Fanuc KAREL source: kb00125.KL

PROGRAM KB00125
%STACKSIZE=65535
%PRIORITY=65535
%NOLOCKGROUP
VAR
P1 : STRING[80]
P2 : INTEGER
BEGIN
P1='A'
P2=1
MSG_DISCO(P1,P2)
END KB00125
